FUNCTION_BLOCK POU EXTENDS FB_AbstructFuture
VAR_INPUT
END_VAR
VAR_OUTPUT
END_VAR
VAR
END_VAR

// NETWORK 1

END_FUNCTION_BLOCK

(* stored: Version 1.1.0.1, ProductVersion 3.1.4024.12
   POU POU: Id {4c1e096a-5673-4fe9-8cc0-66b0c7d97bc7}, SpecialFunc None *)
